# EPICS autosave request: ioc/prj/prjApp/Db/desc_val_settings.req
# FILE... desc_val_settings.req
# USAGE... any record, DESC and VAL fields autosave'd.
$(P).DESC
$(P).VAL
